(* IEC 61131-3 sources: eCockpitGit/test_project/src/%F%00 Library/%F%Common Functions/%F%Networking/%POU%FB_SHA1, 5 files *)

(* ---- %METH%input.st ---- *)
//This method is for inputting a stirng into the function block
// |**Version**|**Author**| **Date** |**Changes**
// | 1         | NSN      | 19-05-20 | Creation
METHOD input
VAR_INPUT
	str		:POINTER TO BYTE;
	len		:DWORD;
END_VAR

(*%!%__DELIMITER__%!%*)
WHILE len > 0 AND NOT(corrupted) DO
	len					:=		len - 1;
	block[index]		:=		str^ AND 16#FF;
	index				:=		index + 1;
	lenLow				:=		lenLow + 8;
	IF lenLow = 0 THEN
		lenHigh			:=		lenHigh + 1;
		IF lenHigh = 0 THEN
			corrupted	:=		TRUE;
		END_IF
	END_IF
	IF index = 64 THEN
		PMB();
	END_IF
	str					:=		str + 1;
END_WHILE

(* ---- %METH%padMessage.st ---- *)
// |**Version**|**Author**| **Date** |**Changes**
// | 1         | NSN      | 19-05-20 | Creation
METHOD PROTECTED padMessage
(*%!%__DELIMITER__%!%*)
IF index > 55 THEN
	block[index]		:=		16#80;
	index				:=		index + 1;
	WHILE index < 64 DO
		block[index]	:=		0;
		index			:=		index + 1;
	END_WHILE
	pmb();
	WHILE index < 56 DO
		block[index]	:=		0;
		index			:=		index + 1;
	END_WHILE
ELSE
	block[index]		:=		16#80;
	index				:=		index + 1;
	WHILE index < 56 DO
		block[index]	:=		0;
		index			:=		index + 1;
	END_WHILE
END_IF
block[56]			:=		TO_BYTE(SHR(lenHigh,24));
block[57]			:=		TO_BYTE(SHR(lenHigh,16));
block[58]			:=		TO_BYTE(SHR(lenHigh,8));
block[59]			:=		TO_BYTE(lenHigh);
block[60]			:=		TO_BYTE(SHR(lenLow,24));
block[61]			:=		TO_BYTE(SHR(lenLow,16));
block[62]			:=		TO_BYTE(SHR(lenLow,8));
block[63]			:=		TO_BYTE(lenLow);
pmb();

(* ---- %METH%pmb.st ---- *)
// |**Version**|**Author**| **Date** |**Changes**
// | 1         | NSN      | 19-05-20 | Creation
METHOD PROTECTED pmb
VAR
	k			:ARRAY[0..3] OF DWORD := [16#5A827999,16#6ED9EBA1,16#8F1BBCDC,16#CA62C1D6];
	t			:INT;
	temp		:DWORD;
	w			:ARRAY[0..79] OF DWORD;
	a,b,c,d,e	:DWORD;
END_VAR
(*%!%__DELIMITER__%!%*)
FOR t := 0 TO 15 DO
	w[t]	:=		SHL(TO_DWORD(block[t * 4]),24);
	w[t]	:=		w[t] OR SHL(TO_DWORD(block[t * 4 + 1]),16);
	w[t]	:=		w[t] OR SHL(TO_DWORD(block[t * 4 + 2]),8);
	w[t]	:=		w[t] OR block[t * 4 + 3];
END_FOR
FOR t := 16 TO 79 DO
	w[t]	:=		ROL(w[t - 3] XOR w[t - 8] XOR w[t - 14] XOR w[t - 16],1);
END_FOR
a			:=		hash[0];
b			:=		hash[1];
c			:=		hash[2];
d			:=		hash[3];
e			:=		hash[4];

FOR t := 0 TO 19 DO
	temp	:=		ROL(a,5) + ((b AND c) OR (NOT(b) AND d)) + e + w[t] + k[0];
	e		:=		d;
	d		:=		c;
	c		:=		ROL(b,30);
	b		:=		a;
	a		:=		temp;
END_FOR

FOR t := 20 TO 39 DO
	temp	:=		ROL(a,5) + (b XOR c XOR d) + e + w[t] + k[1];
	e		:=		d;
	d		:=		c;
	c		:=		ROL(b,30);
	b		:=		a;
	a		:=		temp;
END_FOR

FOR t := 40 TO 59 DO
	temp	:=		ROL(a,5) + ((b AND c) OR (b AND d) OR (c AND d)) + e + w[t] + k[2];
	e		:=		d;
	d		:=		c;
	c		:=		ROL(b,30);
	b		:=		a;
	a		:=		temp;
END_FOR

FOR t := 60 TO 79 DO
	temp	:=		ROL(a,5) + (b XOR c XOR d) + e + w[t] + k[3];
	e		:=		d;
	d		:=		c;
	c		:=		ROL(b,30);
	b		:=		a;
	a		:=		temp;
END_FOR

hash[0]		:=		hash[0] + a;
hash[1]		:=		hash[1] + b;
hash[2]		:=		hash[2] + c;
hash[3]		:=		hash[3] + d;
hash[4]		:=		hash[4] + e;

index		:=		0;

(* ---- %METH%result.st ---- *)
//This method returns the result of the hash calculation in bytes
// |**Version**|**Author**| **Date** |**Changes**
// | 1         | NSN      | 19-05-20 | Creation
METHOD result
VAR_INPUT
	output		:POINTER TO ARRAY[0..19] OF BYTE;	//Array of at least 20 bytes
END_VAR
VAR
	i			:UINT;
END_VAR
(*%!%__DELIMITER__%!%*)
IF corrupted THEN
	RETURN;
END_IF
IF NOT(computed) THEN
	padMessage();
	FOR i := 0 TO 63 DO
		block[i]	:=		0;
	END_FOR
	lenLow			:=		0;
	lenHigh			:=		0;
	computed		:=		TRUE;
END_IF
FOR i := 0 TO 19 DO
	output^[i]		:=		TO_BYTE(SHR(hash[SHR(i,2)],8 * (3 - (i AND 16#03))));
END_FOR

(* ---- %METH%resultHex.st ---- *)
//This method returns the result of the hash to a hexadecimal sting
// |**Version**|**Author**| **Date** |**Changes**
// | 1         | NSN      | 19-05-20 | Creation
METHOD resultHex :STRING(40)
VAR
	i			:BYTE;
	digest		:ARRAY[0..19] OF BYTE;
	hexbuffer	:BYTE;
END_VAR
VAR CONSTANT
	hexes		:ARRAY[0..15] OF BYTE := [48,49,50,51,52,53,54,55,56,57,97,98,99,100,101,102];
END_VAR
(*%!%__DELIMITER__%!%*)
result(output:=ADR(digest));
FOR i := 1 TO 20 DO
	hexbuffer			:=		SHR(digest[i-1],4);
	hexbuffer			:=		hexes[hexbuffer];
	resultHex[i*2-2]	:=		hexbuffer;
	hexbuffer			:=		digest[i-1] AND 15;
	hexbuffer			:=		hexes[hexbuffer];
	resultHex[i*2-1]	:=		hexbuffer;
END_FOR
